VAR_GLOBAL
    // Achsen ***************************************************	
	Y_Achse_steuern						: DUT_Achse_Steuern;		
	Y_Achse_status						: DUT_Achse_Status;		

    // Frequenzumrichter ****************************************
	Trans_Bandseite_steuern				: DUT_SEW_FU_Steuern;	
	Trans_Bandseite_status				: DUT_SEW_FU_Status;

    // Ventile **************************************************
    Laengsanschl          				: DUT_Ventil_sps;
    Schienenklemm          				: DUT_Ventil_sps;

    // interne Variablen ****************************************
    sk_Freigabe                         : BOOL;
    sk                                  : INT;
    transport_einfoerdern_bereit        : BOOL;
    transport_ausfoerdern_bereit        : BOOL;

    Tuer_Anwahl                         : BOOL;   // Signal Tür Anwahl, Tür soll geöffnet werden
    Tuer_Freigabe                       : BOOL;   // Signal Tür Freigabe, Tür kann geöffnet werden
END_VAR

(* stored: Version 1.1.0.1
   GVL GVL_3520: Id {b18f0c44-815f-4cdc-b5d5-d3ba4c611616} *)
